{attribute 'qualified_only'}
{attribute 'strict'}
TYPE MC_SYNC_MODE :
(
	enum_member := 0
);
END_TYPE

(* stored: Version 1.1.0.1, ProductVersion 3.1.4024.11
   DUT MC_SYNC_MODE: Id {bd1de811-2c14-49be-9ea5-53066ae55dae} *)
